FUNCTION_BLOCK Tank1_1_1
VAR_INPUT
	//bSwitchFill : BOOL;
	bSwitchSink : BOOL;
END_VAR
VAR_IN_OUT
	bSwitchFill : BOOL;
END_VAR
VAR_OUTPUT
END_VAR
VAR
	bShl : BOOL := FALSE;
	bSll : BOOL := TRUE;
	bS90l : BOOL;
	nState : INT;
	level: INT := 3;
	tTime : TON;
	rTrig : R_TRIG;	
	
END_VAR


IF level < 5 THEN
	bShl := FALSE;	
	bS90l := TRUE;
	bSll := TRUE;
ELSIF level >= 5 AND level < 90 THEN
	bShl := FALSE;	
	bS90l := TRUE;
	bSll := FALSE;
ELSIF level >= 90 AND level < 100 THEN
	bShl := FALSE;	
	bS90l := FALSE;
	bSll := FALSE;
ELSIF level = 100 THEN
	bShl := TRUE;	
	bS90l := FALSE;
	bSll := FALSE;
END_IF




CASE nState OF
	
	0:	
		IF  NOT bSwitchSink THEN
			IF bSll THEN
				bSwitchFill := TRUE;
			END_IF
			tTime(IN := bSwitchFill,PT := T#2S);
			rTrig(CLK := tTime.Q);
			IF rTrig.Q THEN
				level := level + 2;
				tTime(IN := FALSE);
				IF bShl THEN
					bSwitchFill := FALSE;
					nState := 10;
				END_IF
			END_IF
		 		
		ELSE
			IF NOT bSwitchFill THEN
				nState := 10;
			ELSE
				IF bSll THEN
					bSwitchFill := TRUE;
				END_IF
				tTime(IN := bSwitchFill,PT := T#2S);
				rTrig(CLK := tTime.Q);
				IF rTrig.Q THEN
					level := level + 1;
					tTime(IN := FALSE);
					IF bShl THEN
						bSwitchFill := FALSE;
						nState := 10;
					END_IF
				END_IF
			END_IF
		END_IF
		
	10: 
		IF  bSwitchSink THEN
			IF bShl OR NOT bS90l THEN
				bSwitchFill := FALSE;
			ELSE
				bSwitchFill := bSwitchFill;
			END_IF
			IF NOT bSwitchFill THEN
				tTime(IN := bSwitchSink,PT := T#2S);
				rTrig(CLK := tTime.Q);
				IF rTrig.q THEN
					tTime(IN := FALSE);
					level := level - 1;
					IF bSll THEN
						bSwitchSink := FALSE;
						nState := 0;
					END_IF
				END_IF
			ELSE
				nState := 0;
			END_IF
		ELSE
			IF NOT bSwitchFill THEN
				nState := 10;
			ELSE
				nState := 0;
			END_IF		
		END_IF
					
END_CASE

END_FUNCTION_BLOCK

(* stored: Version 1.1.0.1, ProductVersion 3.1.4024.0
   POU Tank1_1_1: Id {0480b423-bb1c-4121-a27e-14f271a2a664}, SpecialFunc None *)
